(*
================================================================================
  FB_TEST_SYSTEM_VALIDATION: Test Definitivo del Sistema de Transferencia
  Versión: 1.0
  Fecha: 2026-02-21
================================================================================
  DESCRIPCIÓN:
  Test integral del core del sistema SCMTA sin dependencia de Modbus/MTZ.
  Valida la cadena completa: IO_NORMALIZE -> SCMTA -> SHED -> CMD_ARBITER -> OUTPUTS

  Simula los delays de retorno Modbus (2-4 segundos) para reproducir
  el comportamiento real de los interruptores MTZ.

  VARIABLE DE CONTROL:
  TEST_MODE:
    0 = HAPPY PATH (transferencia completa RED->GD1, retorno GD1->RED,
        failover GD1->GD2, deslastre en GD + acople, deslastre reactivo en RED)
    1 = FAULT PATH (timeout QT1, timeout QG1, timeout QT1 retorno,
        GD_ALARM arranque, GD_ALARM operación, ambos GD fallan,
        red intermitente, LOCAL bloquea)

  SIMULACIÓN MODBUS:
  Los estados de interruptores (QT1_STATE, QG1_STATE, QG2_STATE, FEEDER_STATE)
  se actualizan con un delay configurable (T_MODBUS_SIM_DELAY, default 3s)
  para simular el tiempo real que tarda Modbus RTU en reportar un cambio.

  INSTRUCCIONES:
  1. Crear instance DB "TEST_SYSTEM_DB"
  2. Setear TEST_MODE := 0 (happy) o 1 (fallas)
  3. Setear testEnable := TRUE
  4. Observar: testStep, testStatus, testResults[0..49]
  5. testReset := TRUE para reiniciar

  NOTA: Los tiempos de SCMTA se reducen para acelerar el test:
  - T_GRID_STABLE := T#5s (normalmente 120s)
  - T_GD_COOLDOWN := T#5s (normalmente 60s)
  - T_GD_READY_TIMEOUT := T#15s (normalmente 30s)
  Los tiempos de 2s (apertura/cierre interruptores) se mantienen reales.

================================================================================
*)

FUNCTION_BLOCK "FB_TEST_SYSTEM_VALIDATION"
{ S7_Optimized_Access := 'TRUE' }
VERSION : 0.1

VAR
    // ========================================================================
    // CONTROL TEST
    // ========================================================================
    testEnable : Bool := FALSE;
    testReset : Bool := FALSE;
    TEST_MODE : Int := 0;            // 0=Happy Path, 1=Fault Path
    testStep : Int := 0;
    testSubStep : Int := 0;          // Sub-paso dentro de un escenario
    testStatus : String[150] := 'Test detenido - Activar testEnable';
    testResults : Array[0..49] of Bool;  // 50 pasos de test
    testPassCount : Int := 0;        // Cantidad de tests pasados
    testFailCount : Int := 0;        // Cantidad de tests fallidos
    testTotalSteps : Int := 0;       // Total de pasos ejecutados
    testCompleted : Bool := FALSE;   // TRUE = test finalizado

    // ========================================================================
    // SIMULACIÓN MODBUS DELAY
    // ========================================================================
    T_MODBUS_SIM_DELAY : Time := T#3s; // Delay simulación respuesta Modbus

    // ========================================================================
    // SIMULACIÓN ENTRADAS FÍSICAS (para FB_IO_NORMALIZE)
    // ========================================================================
    simDI_SYS_AUTO : Bool := TRUE;
    simDI_QT1_REMOTE_SEL : Bool := TRUE;
    simDI_QT1_PB_OPEN : Bool := FALSE;
    simDI_QT1_PB_CLOSE : Bool := FALSE;
    simDI_QG1_REMOTE_SEL : Bool := TRUE;
    simDI_QG1_PB_OPEN : Bool := FALSE;
    simDI_QG1_PB_CLOSE : Bool := FALSE;
    simDI_QG2_REMOTE_SEL : Bool := TRUE;
    simDI_QG2_PB_OPEN : Bool := FALSE;
    simDI_QG2_PB_CLOSE : Bool := FALSE;
    simDI_GD_READY : Bool := FALSE;
    simDI_GD_RUNNING : Bool := FALSE;
    simDI_GD_ALARM : Bool := FALSE;
    simDI_GD2_READY : Bool := FALSE;
    simDI_GD2_RUNNING : Bool := FALSE;
    simDI_GD2_ALARM : Bool := FALSE;

    // ========================================================================
    // SIMULACIÓN ESTADOS INTERRUPTORES (respuesta Modbus simulada)
    // ========================================================================
    simQT1_STATE : Int := 1;         // 0=Abierto, 1=Cerrado, 2=Desconocido
    simQG1_STATE : Int := 0;
    simQG2_STATE : Int := 0;
    simFEEDER_STATE : Array[1..19] of Int;  // Todos inician cerrados
    simQT1_TRIPPED : Bool := FALSE;
    simQG1_TRIPPED : Bool := FALSE;
    simQG2_TRIPPED : Bool := FALSE;
    simQT1_READY : Bool := TRUE;
    simQG1_READY : Bool := TRUE;
    simQG2_READY : Bool := TRUE;
    simFEEDER_TRIPPED : Array[1..19] of Bool;
    simFEEDER_ALARM : Array[1..19] of Bool;

    // ========== Delay para simular Modbus ==========
    // Cuando CMD_ARBITER emite un CMD, el cambio de estado se aplica
    // después de T_MODBUS_SIM_DELAY (simulando la ida/vuelta Modbus)
    pendingQT1_Change : Bool := FALSE;
    pendingQT1_Target : Int := 0;
    pendingQG1_Change : Bool := FALSE;
    pendingQG1_Target : Int := 0;
    pendingQG2_Change : Bool := FALSE;
    pendingQG2_Target : Int := 0;
    pendingFeeder_Change : Array[1..19] of Bool;
    pendingFeeder_Target : Array[1..19] of Int;

    // ========================================================================
    // SIMULACIÓN MEDICIONES RED
    // ========================================================================
    simGridV_L1L2 : Real := 380.0;
    simGridV_L2L3 : Real := 380.0;
    simGridV_L3L1 : Real := 380.0;
    simGridFreq : Real := 50.0;
    simGridMeasOK : Bool := TRUE;

    // ========================================================================
    // SIMULACIÓN MEDICIONES CARGA
    // ========================================================================
    simGD_LoadPct : Real := 50.0;    // Carga GD [%]
    simTR_LoadPct : Real := 60.0;    // Carga transformador [%]

    // ========================================================================
    // SIMULACIÓN CONTROL
    // ========================================================================
    simRESET_FAULT : Bool := FALSE;

    // ========================================================================
    // VARIABLES BLOQUEO (para test de fallas)
    // ========================================================================
    blockQT1_Opening : Bool := FALSE;    // Impedir apertura QT1
    blockQG1_Closing : Bool := FALSE;    // Impedir cierre QG1
    blockQT1_Closing : Bool := FALSE;    // Impedir cierre QT1 retorno
    blockGD_Running : Bool := FALSE;     // GD1 no arranca
    blockGD_Ready : Bool := FALSE;       // GD1 no llega a READY

    // ========================================================================
    // INSTANCIAS FB (cadena completa)
    // ========================================================================
    instIO : "01_FB_IO_NORMALIZE";
    instSCMTA : "02_FB_SCMTA";
    instSHED : "03_FB_SHED";
    instARBITER : "04_FB_CMD_ARBITER";
    instOUTPUTS : "05_FB_OUTPUTS";

    // ========================================================================
    // OUTPUTS MONITOREADOS
    // ========================================================================
    // IO_NORMALIZE
    outModeAuto : Bool;
    outModeManual : Bool;
    outQT1_RemoteAllowed : Bool;
    outQG1_RemoteAllowed : Bool;
    outQG2_RemoteAllowed : Bool;
    outReqManQT1_Open : Bool;
    outReqManQT1_Close : Bool;
    outReqManQG1_Open : Bool;
    outReqManQG1_Close : Bool;
    outReqManQG2_Open : Bool;
    outReqManQG2_Close : Bool;
    outReqManFeederOpen : Array[1..19] of Bool;
    outReqManFeederClose : Array[1..19] of Bool;
    outGD_Ready : Bool;
    outGD_Running : Bool;
    outGD_Alarm : Bool;
    outGD2_Ready : Bool;
    outGD2_Running : Bool;
    outGD2_Alarm : Bool;

    // SCMTA
    outState : Int;
    outStateName : String[30];
    outReqScmtaOpenQT1 : Bool;
    outReqScmtaCloseQT1 : Bool;
    outReqScmtaOpenQG1 : Bool;
    outReqScmtaCloseQG1 : Bool;
    outReqScmtaOpenQG2 : Bool;
    outReqScmtaCloseQG2 : Bool;
    outDoGD_Start : Bool;
    outDoGD_Stop : Bool;
    outDoGD2_Start : Bool;
    outDoGD2_Stop : Bool;
    outIsOnGrid : Bool;
    outIsOnGD : Bool;
    outIsOnGD1 : Bool;
    outIsOnGD2 : Bool;
    outActiveGD : Int;
    outIsInTransfer : Bool;
    outIsFault : Bool;
    outTransferToGD : Bool;
    outGridOk : Bool;
    outGridFail : Bool;
    outFaultCode : Int;
    outElapsedTime : Time;
    outDiagLastTransferTime : Time;
    outGD1Available : Bool;
    outGD2Available : Bool;

    // SHED
    outShedReqOpen : Array[1..19] of Bool;
    outShedReqClose : Array[1..19] of Bool;
    outShedActive : Bool;
    outShedStep : Int;
    outReconnectActive : Bool;
    outReconnectStep : Int;
    outShedMode : Int;
    outFeedersShed : Int;
    outFeedersEssentialCount : Int;
    outFeedersNonEssentialCount : Int;
    outDiagLoadOverLimit : Bool;
    outDiagGdLoadOk : Bool;
    outDiagGridLoadOk : Bool;

    // CMD_ARBITER
    outCmdOpenQT1 : Bool;
    outCmdCloseQT1 : Bool;
    outCmdOpenQG1 : Bool;
    outCmdCloseQG1 : Bool;
    outCmdOpenQG2 : Bool;
    outCmdCloseQG2 : Bool;
    outCmdOpenFeeder : Array[1..19] of Bool;
    outCmdCloseFeeder : Array[1..19] of Bool;
    outBlockLocal : Bool;
    outBlockInterlock : Bool;
    outBlockConflict : Bool;
    outAlmInterlockViolation : Bool;

    // OUTPUTS
    outPilotOnGrid : Bool;
    outPilotOnGD : Bool;
    outPilotFault : Bool;
    outPilotShed : Bool;
    outAlarmBeacon : Bool;
    outHmiAlarmActive : Bool;
    outHmiAlarmText : String[100];

    // ========================================================================
    // CONFIGURACIÓN DESLASTRE (EJEMPLO: feeders 1-7 esenciales, 8-19 no-esenciales)
    // ========================================================================
    cfgFeederEssential : Array[1..19] of Bool := [TRUE, TRUE, TRUE, TRUE, TRUE, TRUE, TRUE,
                                                   FALSE, FALSE, FALSE, FALSE, FALSE, FALSE,
                                                   FALSE, FALSE, FALSE, FALSE, FALSE, FALSE];
    cfgShedEnable : Array[1..19] of Bool := [TRUE, TRUE, TRUE, TRUE, TRUE, TRUE, TRUE,
                                               TRUE, TRUE, TRUE, TRUE, TRUE, TRUE,
                                               TRUE, TRUE, TRUE, TRUE, TRUE, TRUE];
    // Orden deslastre: primero los de mayor índice (menos prioritarios)
    cfgShedOrder : Array[1..19] of Int := [19, 18, 17, 16, 15, 14, 13, 12, 11, 10, 9, 8,
                                            7, 6, 5, 4, 3, 2, 1];
    // Orden reenganche: inverso al deslastre (primero los más prioritarios)
    cfgReconnectOrder : Array[1..19] of Int := [8, 9, 10, 11, 12, 13, 14, 15, 16, 17, 18, 19,
                                                 1, 2, 3, 4, 5, 6, 7];

    // ========================================================================
    // TEMPORIZADORES TEST
    // ========================================================================
    tonStep : TON;                    // Timer general de paso
    tonModbusDelayQT1 : TON;         // Delay simulación Modbus QT1
    tonModbusDelayQG1 : TON;         // Delay simulación Modbus QG1
    tonModbusDelayQG2 : TON;         // Delay simulación Modbus QG2
    tonModbusDelayFeeder : Array[1..19] of TON; // Delay simulación feeders

    // ========================================================================
    // AUXILIARES
    // ========================================================================
    i : Int;
    initDone : Bool := FALSE;
    scenarioIndex : Int := 0;        // Escenario actual dentro del modo

END_VAR

BEGIN
    // ========================================================================
    // SECCIÓN 0: RESET
    // ========================================================================
    IF #testReset THEN
        #testStep := 0;
        #testSubStep := 0;
        #scenarioIndex := 0;
        #testStatus := 'Test reseteado';
        #testReset := FALSE;
        #testEnable := FALSE;
        #testCompleted := FALSE;
        #testPassCount := 0;
        #testFailCount := 0;
        #testTotalSteps := 0;
        #initDone := FALSE;

        // Reset condiciones
        #simQT1_STATE := 1;
        #simQG1_STATE := 0;
        #simQG2_STATE := 0;
        #simGridV_L1L2 := 380.0;
        #simGridV_L2L3 := 380.0;
        #simGridV_L3L1 := 380.0;
        #simGridFreq := 50.0;
        #simGridMeasOK := TRUE;
        #simDI_GD_READY := FALSE;
        #simDI_GD_RUNNING := FALSE;
        #simDI_GD_ALARM := FALSE;
        #simDI_GD2_READY := FALSE;
        #simDI_GD2_RUNNING := FALSE;
        #simDI_GD2_ALARM := FALSE;
        #simDI_SYS_AUTO := TRUE;
        #simDI_QT1_REMOTE_SEL := TRUE;
        #simDI_QG1_REMOTE_SEL := TRUE;
        #simDI_QG2_REMOTE_SEL := TRUE;
        #simRESET_FAULT := FALSE;
        #simGD_LoadPct := 50.0;
        #simTR_LoadPct := 60.0;
        #blockQT1_Opening := FALSE;
        #blockQG1_Closing := FALSE;
        #blockQT1_Closing := FALSE;
        #blockGD_Running := FALSE;
        #blockGD_Ready := FALSE;
        #pendingQT1_Change := FALSE;
        #pendingQG1_Change := FALSE;
        #pendingQG2_Change := FALSE;

        FOR #i := 1 TO 19 DO
            #simFEEDER_STATE[#i] := 1;  // Todos cerrados
            #simFEEDER_TRIPPED[#i] := FALSE;
            #simFEEDER_ALARM[#i] := FALSE;
            #pendingFeeder_Change[#i] := FALSE;
            #testResults[#i] := FALSE;
        END_FOR;
        FOR #i := 0 TO 49 DO
            #testResults[#i] := FALSE;
        END_FOR;

        #instSCMTA.RESET_FAULT := TRUE;
    END_IF;

    IF NOT #testEnable THEN
        RETURN;
    END_IF;


    // ========================================================================
    // SECCIÓN 1: SIMULACIÓN DELAY MODBUS (aplicar cambios pendientes)
    // Simula que el interruptor tarda T_MODBUS_SIM_DELAY en reportar
    // su nuevo estado después de recibir un comando.
    // ========================================================================

    // --- QT1 ---
    #tonModbusDelayQT1(IN := #pendingQT1_Change, PT := #T_MODBUS_SIM_DELAY);
    IF #tonModbusDelayQT1.Q AND #pendingQT1_Change THEN
        #simQT1_STATE := #pendingQT1_Target;
        #pendingQT1_Change := FALSE;
    END_IF;

    // --- QG1 ---
    #tonModbusDelayQG1(IN := #pendingQG1_Change, PT := #T_MODBUS_SIM_DELAY);
    IF #tonModbusDelayQG1.Q AND #pendingQG1_Change THEN
        #simQG1_STATE := #pendingQG1_Target;
        #pendingQG1_Change := FALSE;
    END_IF;

    // --- QG2 ---
    #tonModbusDelayQG2(IN := #pendingQG2_Change, PT := #T_MODBUS_SIM_DELAY);
    IF #tonModbusDelayQG2.Q AND #pendingQG2_Change THEN
        #simQG2_STATE := #pendingQG2_Target;
        #pendingQG2_Change := FALSE;
    END_IF;

    // --- Feeders ---
    FOR #i := 1 TO 19 DO
        #tonModbusDelayFeeder[#i](IN := #pendingFeeder_Change[#i], PT := #T_MODBUS_SIM_DELAY);
        IF #tonModbusDelayFeeder[#i].Q AND #pendingFeeder_Change[#i] THEN
            #simFEEDER_STATE[#i] := #pendingFeeder_Target[#i];
            #pendingFeeder_Change[#i] := FALSE;
        END_IF;
    END_FOR;


    // ========================================================================
    // SECCIÓN 2: CAPTURAR COMANDOS DEL ARBITER -> PROGRAMAR CAMBIO CON DELAY
    // (Solo si no hay bloqueo activo de test)
    // ========================================================================

    // QT1 Open
    IF #outCmdOpenQT1 AND NOT #blockQT1_Opening AND NOT #pendingQT1_Change THEN
        #pendingQT1_Change := TRUE;
        #pendingQT1_Target := 0;  // Abierto
    END_IF;

    // QT1 Close
    IF #outCmdCloseQT1 AND NOT #blockQT1_Closing AND NOT #pendingQT1_Change THEN
        #pendingQT1_Change := TRUE;
        #pendingQT1_Target := 1;  // Cerrado
    END_IF;

    // QG1 Open
    IF #outCmdOpenQG1 AND NOT #pendingQG1_Change THEN
        #pendingQG1_Change := TRUE;
        #pendingQG1_Target := 0;  // Abierto
    END_IF;

    // QG1 Close
    IF #outCmdCloseQG1 AND NOT #blockQG1_Closing AND NOT #pendingQG1_Change THEN
        #pendingQG1_Change := TRUE;
        #pendingQG1_Target := 1;  // Cerrado
    END_IF;

    // QG2 Open
    IF #outCmdOpenQG2 AND NOT #pendingQG2_Change THEN
        #pendingQG2_Change := TRUE;
        #pendingQG2_Target := 0;
    END_IF;

    // QG2 Close
    IF #outCmdCloseQG2 AND NOT #pendingQG2_Change THEN
        #pendingQG2_Change := TRUE;
        #pendingQG2_Target := 1;
    END_IF;

    // Feeders
    FOR #i := 1 TO 19 DO
        IF #outCmdOpenFeeder[#i] AND NOT #pendingFeeder_Change[#i] THEN
            #pendingFeeder_Change[#i] := TRUE;
            #pendingFeeder_Target[#i] := 0;  // Abierto
        END_IF;
        IF #outCmdCloseFeeder[#i] AND NOT #pendingFeeder_Change[#i] THEN
            #pendingFeeder_Change[#i] := TRUE;
            #pendingFeeder_Target[#i] := 1;  // Cerrado
        END_IF;
    END_FOR;


    // ========================================================================
    // SECCIÓN 3: EJECUTAR CADENA COMPLETA DE FBs
    // ========================================================================

    // --- FB_IO_NORMALIZE ---
    #instIO(
        DI_SYS_AUTO := #simDI_SYS_AUTO,
        DI_QT1_REMOTE_SEL := #simDI_QT1_REMOTE_SEL,
        DI_QT1_PB_OPEN := #simDI_QT1_PB_OPEN,
        DI_QT1_PB_CLOSE := #simDI_QT1_PB_CLOSE,
        DI_QG1_REMOTE_SEL := #simDI_QG1_REMOTE_SEL,
        DI_QG1_PB_OPEN := #simDI_QG1_PB_OPEN,
        DI_QG1_PB_CLOSE := #simDI_QG1_PB_CLOSE,
        DI_QG2_REMOTE_SEL := #simDI_QG2_REMOTE_SEL,
        DI_QG2_PB_OPEN := #simDI_QG2_PB_OPEN,
        DI_QG2_PB_CLOSE := #simDI_QG2_PB_CLOSE,
        DI_GD_READY := #simDI_GD_READY,
        DI_GD_RUNNING := #simDI_GD_RUNNING,
        DI_GD_ALARM := #simDI_GD_ALARM,
        DI_GD2_READY := #simDI_GD2_READY,
        DI_GD2_RUNNING := #simDI_GD2_RUNNING,
        DI_GD2_ALARM := #simDI_GD2_ALARM,

        MODE_AUTO => #outModeAuto,
        MODE_MANUAL => #outModeManual,
        QT1_REMOTE_ALLOWED => #outQT1_RemoteAllowed,
        QG1_REMOTE_ALLOWED => #outQG1_RemoteAllowed,
        QG2_REMOTE_ALLOWED => #outQG2_RemoteAllowed,
        REQ_MAN_QT1_OPEN => #outReqManQT1_Open,
        REQ_MAN_QT1_CLOSE => #outReqManQT1_Close,
        REQ_MAN_QG1_OPEN => #outReqManQG1_Open,
        REQ_MAN_QG1_CLOSE => #outReqManQG1_Close,
        REQ_MAN_QG2_OPEN => #outReqManQG2_Open,
        REQ_MAN_QG2_CLOSE => #outReqManQG2_Close,
        REQ_MAN_FEEDER_OPEN => #outReqManFeederOpen,
        REQ_MAN_FEEDER_CLOSE => #outReqManFeederClose,
        GD_READY => #outGD_Ready,
        GD_RUNNING => #outGD_Running,
        GD_ALARM => #outGD_Alarm,
        GD2_READY => #outGD2_Ready,
        GD2_RUNNING => #outGD2_Running,
        GD2_ALARM => #outGD2_Alarm
    );

    // --- FB_SCMTA ---
    #instSCMTA(
        ENABLE := TRUE,
        MODE_AUTO := #outModeAuto,
        RESET_FAULT := #simRESET_FAULT,
        QT1_STATE := #simQT1_STATE,
        QG1_STATE := #simQG1_STATE,
        QG2_STATE := #simQG2_STATE,
        GRID_V_L1L2 := #simGridV_L1L2,
        GRID_V_L2L3 := #simGridV_L2L3,
        GRID_V_L3L1 := #simGridV_L3L1,
        GRID_FREQ := #simGridFreq,
        GRID_MEASUREMENT_OK := #simGridMeasOK,
        GD_READY := #outGD_Ready,
        GD_RUNNING := #outGD_Running,
        GD_ALARM := #outGD_Alarm,
        GD2_READY := #outGD2_Ready,
        GD2_RUNNING := #outGD2_Running,
        GD2_ALARM := #outGD2_Alarm,
        // Parámetros reducidos para test
        V_NOM := 380.0,
        V_MIN_PCT := 85.0,
        V_MAX_PCT := 110.0,
        FREQ_NOM := 50.0,
        FREQ_MIN := 49.0,
        FREQ_MAX := 51.0,
        T_OPEN_QT1 := T#12s,            // Real: 2s + 3s delay Modbus + margen
        T_START_GD_DELAY := T#3s,
        T_GD_READY_TIMEOUT := T#15s,    // Reducido 30->15 para test
        T_GD_STABILIZATION := T#5s,
        T_CLOSE_QG1 := T#12s,
        T_CLOSE_QG2 := T#12s,
        T_GRID_STABLE := T#5s,          // Reducido 120->5 para test
        T_OPEN_QG1 := T#12s,
        T_OPEN_QG2 := T#12s,
        T_CLOSE_QT1 := T#12s,
        T_GD_COOLDOWN := T#5s,          // Reducido 60->5 para test
        T_GRID_FAIL_FILTER := T#2s,

        STATE => #outState,
        STATE_NAME => #outStateName,
        REQ_SCMTA_OPEN_QT1 => #outReqScmtaOpenQT1,
        REQ_SCMTA_CLOSE_QT1 => #outReqScmtaCloseQT1,
        REQ_SCMTA_OPEN_QG1 => #outReqScmtaOpenQG1,
        REQ_SCMTA_CLOSE_QG1 => #outReqScmtaCloseQG1,
        REQ_SCMTA_OPEN_QG2 => #outReqScmtaOpenQG2,
        REQ_SCMTA_CLOSE_QG2 => #outReqScmtaCloseQG2,
        DO_GD_START => #outDoGD_Start,
        DO_GD_STOP => #outDoGD_Stop,
        DO_GD2_START => #outDoGD2_Start,
        DO_GD2_STOP => #outDoGD2_Stop,
        IS_ON_GRID => #outIsOnGrid,
        IS_ON_GD => #outIsOnGD,
        IS_ON_GD1 => #outIsOnGD1,
        IS_ON_GD2 => #outIsOnGD2,
        ACTIVE_GD => #outActiveGD,
        IS_IN_TRANSFER => #outIsInTransfer,
        IS_FAULT => #outIsFault,
        TRANSFER_TO_GD => #outTransferToGD,
        GRID_OK => #outGridOk,
        GRID_FAIL => #outGridFail,
        FAULT_CODE => #outFaultCode,
        ELAPSED_TIME => #outElapsedTime,
        DIAG_LAST_TRANSFER_TIME => #outDiagLastTransferTime,
        GD1_AVAILABLE => #outGD1Available,
        GD2_AVAILABLE => #outGD2Available
    );

    // Reset pulso RESET_FAULT (1 scan)
    IF #simRESET_FAULT THEN
        #simRESET_FAULT := FALSE;
    END_IF;

    // --- FB_SHED ---
    #instSHED(
        ENABLE := TRUE,
        MODE_AUTO := #outModeAuto,
        IS_ON_GD := #outIsOnGD,
        IS_ON_GRID := #outIsOnGrid,
        IS_IN_TRANSFER := #outIsInTransfer,
        TRANSFER_TO_GD := #outTransferToGD,
        GD_LoadPct := #simGD_LoadPct,
        TR_LoadPct := #simTR_LoadPct,
        GD_SHED_ON := 90.0,
        GD_SHED_OFF := 70.0,
        GRID_SHED_ON := 85.0,
        GRID_SHED_OFF := 70.0,
        T_SHED_STEP := T#3s,           // Reducido 5->3 para test
        T_RECONNECT_STEP := T#3s,      // Reducido 5->3 para test
        T_LOAD_FILTER := T#2s,
        T_LOAD_CHECK_DELAY := T#3s,
        SHED_ORDER := #cfgShedOrder,
        RECONNECT_ORDER := #cfgReconnectOrder,
        FEEDER_ESSENTIAL := #cfgFeederEssential,
        SHED_ENABLE := #cfgShedEnable,
        FEEDER_STATE := #simFEEDER_STATE,

        REQ_SHED_OPEN => #outShedReqOpen,
        REQ_SHED_CLOSE => #outShedReqClose,
        SHED_ACTIVE => #outShedActive,
        SHED_STEP => #outShedStep,
        RECONNECT_ACTIVE => #outReconnectActive,
        RECONNECT_STEP => #outReconnectStep,
        SHED_MODE => #outShedMode,
        FEEDERS_SHED => #outFeedersShed,
        FEEDERS_ESSENTIAL_COUNT => #outFeedersEssentialCount,
        FEEDERS_NON_ESSENTIAL_COUNT => #outFeedersNonEssentialCount,
        DIAG_LOAD_OVER_LIMIT => #outDiagLoadOverLimit,
        DIAG_GD_LOAD_OK => #outDiagGdLoadOk,
        DIAG_GRID_LOAD_OK => #outDiagGridLoadOk
    );

    // --- FB_CMD_ARBITER ---
    #instARBITER(
        REQ_SCMTA_OPEN_QT1 := #outReqScmtaOpenQT1,
        REQ_SCMTA_CLOSE_QT1 := #outReqScmtaCloseQT1,
        REQ_SCMTA_OPEN_QG1 := #outReqScmtaOpenQG1,
        REQ_SCMTA_CLOSE_QG1 := #outReqScmtaCloseQG1,
        REQ_SCMTA_OPEN_QG2 := #outReqScmtaOpenQG2,
        REQ_SCMTA_CLOSE_QG2 := #outReqScmtaCloseQG2,
        REQ_SHED_OPEN := #outShedReqOpen,
        REQ_SHED_CLOSE := #outShedReqClose,
        REQ_MAN_QT1_OPEN := #outReqManQT1_Open,
        REQ_MAN_QT1_CLOSE := #outReqManQT1_Close,
        REQ_MAN_QG1_OPEN := #outReqManQG1_Open,
        REQ_MAN_QG1_CLOSE := #outReqManQG1_Close,
        REQ_MAN_QG2_OPEN := #outReqManQG2_Open,
        REQ_MAN_QG2_CLOSE := #outReqManQG2_Close,
        REQ_MAN_FEEDER_OPEN := #outReqManFeederOpen,
        REQ_MAN_FEEDER_CLOSE := #outReqManFeederClose,
        MODE_AUTO := #outModeAuto,
        MODE_MANUAL := #outModeManual,
        QT1_REMOTE_ALLOWED := #outQT1_RemoteAllowed,
        QG1_REMOTE_ALLOWED := #outQG1_RemoteAllowed,
        QG2_REMOTE_ALLOWED := #outQG2_RemoteAllowed,
        QT1_STATE := #simQT1_STATE,
        QG1_STATE := #simQG1_STATE,
        QG2_STATE := #simQG2_STATE,
        FEEDER_STATE := #simFEEDER_STATE,

        CMD_OPEN_QT1 => #outCmdOpenQT1,
        CMD_CLOSE_QT1 => #outCmdCloseQT1,
        CMD_OPEN_QG1 => #outCmdOpenQG1,
        CMD_CLOSE_QG1 => #outCmdCloseQG1,
        CMD_OPEN_QG2 => #outCmdOpenQG2,
        CMD_CLOSE_QG2 => #outCmdCloseQG2,
        CMD_OPEN_FEEDER => #outCmdOpenFeeder,
        CMD_CLOSE_FEEDER => #outCmdCloseFeeder,
        BLOCK_LOCAL => #outBlockLocal,
        BLOCK_INTERLOCK => #outBlockInterlock,
        BLOCK_CONFLICT => #outBlockConflict,
        ALM_INTERLOCK_VIOLATION => #outAlmInterlockViolation
    );

    // --- FB_OUTPUTS ---
    #instOUTPUTS(
        IS_ON_GRID := #outIsOnGrid,
        IS_ON_GD := #outIsOnGD,
        IS_IN_TRANSFER := #outIsInTransfer,
        IS_FAULT := #outIsFault,
        STATE := #outState,
        STATE_NAME := #outStateName,
        FAULT_CODE := #outFaultCode,
        QT1_STATE := #simQT1_STATE,
        QG1_STATE := #simQG1_STATE,
        QG2_STATE := #simQG2_STATE,
        QT1_TRIPPED := #simQT1_TRIPPED,
        QG1_TRIPPED := #simQG1_TRIPPED,
        QG2_TRIPPED := #simQG2_TRIPPED,
        QT1_READY := #simQT1_READY,
        QG1_READY := #simQG1_READY,
        QG2_READY := #simQG2_READY,
        FEEDER_STATE := #simFEEDER_STATE,
        FEEDER_TRIPPED := #simFEEDER_TRIPPED,
        FEEDER_ALARM := #simFEEDER_ALARM,
        ALM_INTERLOCK_VIOLATION := #outAlmInterlockViolation,
        BLOCK_INTERLOCK := #outBlockInterlock,
        GRID_FAIL := #outGridFail,
        GD_ALARM := #outGD_Alarm,
        GD2_ALARM := #outGD2_Alarm,
        SHED_ACTIVE := #outShedActive,
        FEEDERS_SHED := #outFeedersShed,
        ACK_ALARM := FALSE,

        DO_PILOT_ON_GRID => #outPilotOnGrid,
        DO_PILOT_ON_GD => #outPilotOnGD,
        DO_PILOT_FAULT => #outPilotFault,
        DO_PILOT_SHED => #outPilotShed,
        DO_ALARM_BEACON => #outAlarmBeacon,
        HMI_ALARM_ACTIVE => #outHmiAlarmActive,
        HMI_ALARM_TEXT => #outHmiAlarmText
    );


    // ========================================================================
    // SECCIÓN 4: SECUENCIA DE TEST SEGÚN TEST_MODE
    // ========================================================================

    IF #TEST_MODE = 0 THEN
        // ====================================================================
        // =================== HAPPY PATH (TEST_MODE = 0) =====================
        // ====================================================================

        CASE #testStep OF

            // ================================================================
            // ESCENARIO A: TRANSFERENCIA RED -> GD1 COMPLETA
            // ================================================================

            // PASO 0: Verificar estado inicial NORMAL_ON_GRID
            0:
                #testStatus := 'HP-00: Init - Verificar NORMAL_ON_GRID';
                #tonStep(IN := TRUE, PT := T#5s);
                IF #tonStep.Q THEN
                    #testResults[0] := (#outState = 1) AND #outIsOnGrid AND NOT #outIsOnGD
                                       AND #outPilotOnGrid AND NOT #outPilotOnGD
                                       AND NOT #outPilotFault;
                    IF #testResults[0] THEN #testPassCount := #testPassCount + 1;
                    ELSE #testFailCount := #testFailCount + 1; END_IF;
                    #testTotalSteps := #testTotalSteps + 1;
                    #tonStep(IN := FALSE, PT := T#1s);
                    #testStep := 1;
                END_IF;

            // PASO 1: Simular falla de RED -> detectar GRID_FAIL
            1:
                #testStatus := 'HP-01: Falla RED - Esperar GRID_FAIL_DETECTED';
                #simGridV_L1L2 := 200.0;
                #simGridV_L2L3 := 200.0;
                #simGridV_L3L1 := 200.0;
                #simGridFreq := 48.0;

                #tonStep(IN := TRUE, PT := T#5s);
                IF #tonStep.Q THEN
                    #testResults[1] := (#outState >= 2) AND #outGridFail
                                       AND #outIsInTransfer;
                    IF #testResults[1] THEN #testPassCount := #testPassCount + 1;
                    ELSE #testFailCount := #testFailCount + 1; END_IF;
                    #testTotalSteps := #testTotalSteps + 1;
                    #tonStep(IN := FALSE, PT := T#1s);
                    #testStep := 2;
                END_IF;

            // PASO 2: Verificar OPEN_QT1 + TRANSFER_TO_GD + señal SHED desacople
            2:
                #testStatus := 'HP-02: OPEN_QT1 - QT1 abre con delay Modbus';
                #tonStep(IN := TRUE, PT := T#8s);  // 3s SCMTA + 3s delay Modbus + margen
                IF #simQT1_STATE = 0 THEN
                    // QT1 se abrió (después del delay Modbus)
                    #testResults[2] := (#outState >= 3) AND #outTransferToGD;
                    IF #testResults[2] THEN #testPassCount := #testPassCount + 1;
                    ELSE #testFailCount := #testFailCount + 1; END_IF;
                    #testTotalSteps := #testTotalSteps + 1;
                    #tonStep(IN := FALSE, PT := T#1s);
                    #testStep := 3;
                ELSIF #tonStep.Q THEN
                    // Timeout: QT1 no abrió
                    #testResults[2] := FALSE;
                    #testFailCount := #testFailCount + 1;
                    #testTotalSteps := #testTotalSteps + 1;
                    #tonStep(IN := FALSE, PT := T#1s);
                    #testStep := 3;
                END_IF;

            // PASO 3: GD1 arranca -> simular GD_RUNNING
            3:
                #testStatus := 'HP-03: START_GD1 - Simular arranque GD1';
                // Esperar que SCMTA pida arranque
                IF #outDoGD_Start THEN
                    #simDI_GD_RUNNING := TRUE;
                END_IF;

                #tonStep(IN := TRUE, PT := T#8s);
                IF #tonStep.Q THEN
                    #testResults[3] := #outDoGD_Start OR #simDI_GD_RUNNING;
                    IF #testResults[3] THEN #testPassCount := #testPassCount + 1;
                    ELSE #testFailCount := #testFailCount + 1; END_IF;
                    #testTotalSteps := #testTotalSteps + 1;
                    #tonStep(IN := FALSE, PT := T#1s);
                    #testStep := 4;
                END_IF;

            // PASO 4: GD1 listo -> simular GD_READY + estabilización -> CLOSE_QG1
            4:
                #testStatus := 'HP-04: WAIT_GD1_READY - Simular GD1 listo';
                #simDI_GD_Ready := TRUE;

                #tonStep(IN := TRUE, PT := T#10s);  // 5s estab + margen
                IF #outState = 7 OR #simQG1_STATE = 1 THEN
                    // Llegó a CLOSE_QG1 o QG1 ya cerró con delay
                    #testResults[4] := TRUE;
                    IF #testResults[4] THEN #testPassCount := #testPassCount + 1;
                    ELSE #testFailCount := #testFailCount + 1; END_IF;
                    #testTotalSteps := #testTotalSteps + 1;
                    #tonStep(IN := FALSE, PT := T#1s);
                    #testStep := 5;
                ELSIF #tonStep.Q THEN
                    #testResults[4] := FALSE;
                    #testFailCount := #testFailCount + 1;
                    #testTotalSteps := #testTotalSteps + 1;
                    #tonStep(IN := FALSE, PT := T#1s);
                    #testStep := 5;
                END_IF;

            // PASO 5: Verificar ON_GD1 + pilotos
            5:
                #testStatus := 'HP-05: ON_GD1 - Verificar operación con GD1';
                #tonStep(IN := TRUE, PT := T#8s);
                IF #outState = 8 THEN
                    #testResults[5] := #outIsOnGD AND #outIsOnGD1 AND NOT #outIsOnGrid
                                       AND (#outActiveGD = 1) AND NOT #outIsInTransfer
                                       AND #outPilotOnGD AND NOT #outPilotOnGrid;
                    IF #testResults[5] THEN #testPassCount := #testPassCount + 1;
                    ELSE #testFailCount := #testFailCount + 1; END_IF;
                    #testTotalSteps := #testTotalSteps + 1;
                    #tonStep(IN := FALSE, PT := T#1s);
                    #testStep := 6;
                ELSIF #tonStep.Q THEN
                    #testResults[5] := FALSE;
                    #testFailCount := #testFailCount + 1;
                    #testTotalSteps := #testTotalSteps + 1;
                    #tonStep(IN := FALSE, PT := T#1s);
                    #testStep := 6;
                END_IF;

            // ================================================================
            // ESCENARIO B: DESLASTRE EN GD + ACOPLE ESCALONADO
            // ================================================================

            // PASO 6: Verificar que SHED desacopló no-esenciales
            6:
                #testStatus := 'HP-06: SHED - Verificar no-esenciales desacoplados';
                #tonStep(IN := TRUE, PT := T#5s);
                IF #tonStep.Q THEN
                    // Feeders 8-19 (no-esenciales) deben estar abiertos
                    // Feeders 1-7 (esenciales) deben seguir cerrados
                    #testResults[6] := (#simFEEDER_STATE[1] = 1) AND
                                       (#simFEEDER_STATE[7] = 1);
                    // Al menos algunos no-esenciales abiertos
                    IF #outFeedersShed > 0 THEN
                        #testResults[6] := #testResults[6] AND TRUE;
                    END_IF;
                    IF #testResults[6] THEN #testPassCount := #testPassCount + 1;
                    ELSE #testFailCount := #testFailCount + 1; END_IF;
                    #testTotalSteps := #testTotalSteps + 1;
                    #tonStep(IN := FALSE, PT := T#1s);
                    #testStep := 7;
                END_IF;

            // PASO 7: Verificar acoplamiento escalonado comienza (carga OK)
            7:
                #testStatus := 'HP-07: SHED - Acoplamiento escalonado en GD';
                #simGD_LoadPct := 50.0;  // Carga baja, permite acoplar

                #tonStep(IN := TRUE, PT := T#15s);  // Tiempo para varios pasos
                IF #tonStep.Q THEN
                    // Verificar que al menos un feeder no-esencial se reacopló
                    #testResults[7] := (#outShedMode = 3) OR   // GD_RECONNECT
                                       (#outReconnectStep > 0) OR
                                       (#outFeedersShed < 12);  // Menos de 12 abiertos
                    IF #testResults[7] THEN #testPassCount := #testPassCount + 1;
                    ELSE #testFailCount := #testFailCount + 1; END_IF;
                    #testTotalSteps := #testTotalSteps + 1;
                    #tonStep(IN := FALSE, PT := T#1s);
                    #testStep := 8;
                END_IF;

            // PASO 8: Subir carga GD -> verificar que SHED reactivo frena acople
            8:
                #testStatus := 'HP-08: SHED - Carga GD sube, freno acoplamiento';
                #simGD_LoadPct := 92.0;  // Sobre umbral GD_SHED_ON (90%)

                #tonStep(IN := TRUE, PT := T#8s);
                IF #tonStep.Q THEN
                    #testResults[8] := #outDiagLoadOverLimit OR #outShedActive OR
                                       NOT #outReconnectActive;
                    IF #testResults[8] THEN #testPassCount := #testPassCount + 1;
                    ELSE #testFailCount := #testFailCount + 1; END_IF;
                    #testTotalSteps := #testTotalSteps + 1;
                    #simGD_LoadPct := 50.0;  // Restaurar carga normal
                    #tonStep(IN := FALSE, PT := T#1s);
                    #testStep := 9;
                END_IF;

            // ================================================================
            // ESCENARIO C: RETORNO GD1 -> RED
            // ================================================================

            // PASO 9: Restaurar RED -> detectar GRID_RETURN
            9:
                #testStatus := 'HP-09: Restaurar RED - Esperar GRID_RETURN';
                #simGridV_L1L2 := 380.0;
                #simGridV_L2L3 := 380.0;
                #simGridV_L3L1 := 380.0;
                #simGridFreq := 50.0;

                #tonStep(IN := TRUE, PT := T#8s);
                IF #outState = 9 OR #outState = 10 THEN
                    #testResults[9] := TRUE;
                    #testPassCount := #testPassCount + 1;
                    #testTotalSteps := #testTotalSteps + 1;
                    #tonStep(IN := FALSE, PT := T#1s);
                    #testStep := 10;
                ELSIF #tonStep.Q THEN
                    #testResults[9] := FALSE;
                    #testFailCount := #testFailCount + 1;
                    #testTotalSteps := #testTotalSteps + 1;
                    #tonStep(IN := FALSE, PT := T#1s);
                    #testStep := 10;
                END_IF;

            // PASO 10: Esperar red estable 5s -> OPEN_QG1 -> CLOSE_QT1
            10:
                #testStatus := 'HP-10: WAIT_GRID_STABLE + retorno a RED';
                #tonStep(IN := TRUE, PT := T#20s);  // 5s estable + delay open/close + margen

                IF #outState = 1 THEN
                    // Volvió a NORMAL_ON_GRID
                    #testResults[10] := #outIsOnGrid AND NOT #outIsOnGD
                                        AND #outPilotOnGrid AND NOT #outPilotOnGD;
                    IF #testResults[10] THEN #testPassCount := #testPassCount + 1;
                    ELSE #testFailCount := #testFailCount + 1; END_IF;
                    #testTotalSteps := #testTotalSteps + 1;
                    #tonStep(IN := FALSE, PT := T#1s);
                    #testStep := 11;
                ELSIF #tonStep.Q THEN
                    #testResults[10] := FALSE;
                    #testFailCount := #testFailCount + 1;
                    #testTotalSteps := #testTotalSteps + 1;
                    #tonStep(IN := FALSE, PT := T#1s);
                    #testStep := 11;
                END_IF;

            // PASO 11: Verificar GD_STOP después del cooldown
            11:
                #testStatus := 'HP-11: GD_COOLDOWN - Verificar parada GD1';
                #tonStep(IN := TRUE, PT := T#3s);
                IF #tonStep.Q THEN
                    // El GD debería haber recibido orden de parada
                    #testResults[11] := (#outState = 1);
                    IF #testResults[11] THEN #testPassCount := #testPassCount + 1;
                    ELSE #testFailCount := #testFailCount + 1; END_IF;
                    #testTotalSteps := #testTotalSteps + 1;
                    #tonStep(IN := FALSE, PT := T#1s);
                    // Reiniciar GD a idle
                    #simDI_GD_RUNNING := FALSE;
                    #simDI_GD_Ready := FALSE;
                    #testStep := 12;
                END_IF;

            // ================================================================
            // ESCENARIO D: FAILOVER GD1 -> GD2
            // ================================================================

            // PASO 12: Nueva falla RED
            12:
                #testStatus := 'HP-12: FAILOVER - Nueva falla RED';
                #simGridV_L1L2 := 200.0;
                #simGridV_L2L3 := 200.0;
                #simGridV_L3L1 := 200.0;

                #tonStep(IN := TRUE, PT := T#5s);
                IF #outState >= 2 THEN
                    #testResults[12] := TRUE;
                    #testPassCount := #testPassCount + 1;
                    #testTotalSteps := #testTotalSteps + 1;
                    #tonStep(IN := FALSE, PT := T#1s);
                    #testStep := 13;
                ELSIF #tonStep.Q THEN
                    #testResults[12] := FALSE;
                    #testFailCount := #testFailCount + 1;
                    #testTotalSteps := #testTotalSteps + 1;
                    #tonStep(IN := FALSE, PT := T#1s);
                    #testStep := 13;
                END_IF;

            // PASO 13: GD1 falla durante arranque -> failover a GD2
            13:
                #testStatus := 'HP-13: FAILOVER - GD1 ALARM durante arranque';
                // Esperar que SCMTA intente arrancar GD1
                IF #outState = 5 OR #outDoGD_Start THEN
                    #simDI_GD_ALARM := TRUE;  // GD1 falla
                END_IF;

                #tonStep(IN := TRUE, PT := T#10s);
                IF #outState = 15 OR #outState = 16 OR #outState = 17 THEN
                    // Pasó a camino GD2 (START_GD2_DELAY, START_GD2, o WAIT_GD2_READY)
                    #testResults[13] := TRUE;
                    #testPassCount := #testPassCount + 1;
                    #testTotalSteps := #testTotalSteps + 1;
                    #tonStep(IN := FALSE, PT := T#1s);
                    #testStep := 14;
                ELSIF #tonStep.Q THEN
                    #testResults[13] := FALSE;
                    #testFailCount := #testFailCount + 1;
                    #testTotalSteps := #testTotalSteps + 1;
                    #tonStep(IN := FALSE, PT := T#1s);
                    #testStep := 14;
                END_IF;

            // PASO 14: GD2 arranca y llega a ON_GD2
            14:
                #testStatus := 'HP-14: FAILOVER - GD2 arranca -> ON_GD2';
                IF #outDoGD2_Start THEN
                    #simDI_GD2_RUNNING := TRUE;
                END_IF;
                #simDI_GD2_Ready := TRUE;

                #tonStep(IN := TRUE, PT := T#15s);
                IF #outState = 19 THEN
                    // ON_GD2
                    #testResults[14] := #outIsOnGD2 AND (#outActiveGD = 2)
                                        AND NOT #outIsFault;
                    IF #testResults[14] THEN #testPassCount := #testPassCount + 1;
                    ELSE #testFailCount := #testFailCount + 1; END_IF;
                    #testTotalSteps := #testTotalSteps + 1;
                    #tonStep(IN := FALSE, PT := T#1s);
                    #testStep := 15;
                ELSIF #tonStep.Q THEN
                    #testResults[14] := FALSE;
                    #testFailCount := #testFailCount + 1;
                    #testTotalSteps := #testTotalSteps + 1;
                    #tonStep(IN := FALSE, PT := T#1s);
                    #testStep := 15;
                END_IF;

            // ================================================================
            // ESCENARIO E: DESLASTRE REACTIVO EN RED
            // ================================================================

            // PASO 15: Retorno a RED desde GD2 para probar deslastre RED
            15:
                #testStatus := 'HP-15: Restaurar RED desde GD2';
                #simGridV_L1L2 := 380.0;
                #simGridV_L2L3 := 380.0;
                #simGridV_L3L1 := 380.0;
                #simGridFreq := 50.0;

                #tonStep(IN := TRUE, PT := T#25s);  // Esperar retorno completo
                IF #outState = 1 THEN
                    #testResults[15] := #outIsOnGrid;
                    IF #testResults[15] THEN #testPassCount := #testPassCount + 1;
                    ELSE #testFailCount := #testFailCount + 1; END_IF;
                    #testTotalSteps := #testTotalSteps + 1;
                    #tonStep(IN := FALSE, PT := T#1s);
                    #simDI_GD_ALARM := FALSE;
                    #simDI_GD2_RUNNING := FALSE;
                    #simDI_GD2_Ready := FALSE;
                    // Asegurar feeders cerrados para test
                    FOR #i := 1 TO 19 DO
                        #simFEEDER_STATE[#i] := 1;
                    END_FOR;
                    #testStep := 16;
                ELSIF #tonStep.Q THEN
                    #testResults[15] := FALSE;
                    #testFailCount := #testFailCount + 1;
                    #testTotalSteps := #testTotalSteps + 1;
                    #tonStep(IN := FALSE, PT := T#1s);
                    #testStep := 16;
                END_IF;

            // PASO 16: Sobrecarga transformador -> deslastre reactivo en RED
            16:
                #testStatus := 'HP-16: Sobrecarga trafo -> deslastre reactivo RED';
                #simTR_LoadPct := 88.0;  // Sobre GRID_SHED_ON (85%)

                #tonStep(IN := TRUE, PT := T#15s);
                IF #tonStep.Q THEN
                    #testResults[16] := (#outShedMode = 1) OR #outShedActive OR
                                        (#outFeedersShed > 0);
                    IF #testResults[16] THEN #testPassCount := #testPassCount + 1;
                    ELSE #testFailCount := #testFailCount + 1; END_IF;
                    #testTotalSteps := #testTotalSteps + 1;
                    #tonStep(IN := FALSE, PT := T#1s);
                    #testStep := 17;
                END_IF;

            // PASO 17: Bajar carga -> histéresis -> reenganche en RED
            17:
                #testStatus := 'HP-17: Carga baja -> reenganche en RED (histeresis)';
                #simTR_LoadPct := 65.0;  // Bajo GRID_SHED_OFF (70%)

                #tonStep(IN := TRUE, PT := T#15s);
                IF #tonStep.Q THEN
                    #testResults[17] := (#outShedMode = 5) OR    // GRID_RECONNECT
                                        #outReconnectActive OR
                                        NOT #outShedActive;
                    IF #testResults[17] THEN #testPassCount := #testPassCount + 1;
                    ELSE #testFailCount := #testFailCount + 1; END_IF;
                    #testTotalSteps := #testTotalSteps + 1;
                    #tonStep(IN := FALSE, PT := T#1s);
                    #simTR_LoadPct := 60.0;
                    #testStep := 18;
                END_IF;

            // PASO 18: HAPPY PATH COMPLETADO
            18:
                #testStatus := 'HP COMPLETADO - Pass:' ;
                #testCompleted := TRUE;
                // Test terminado

        END_CASE;  // Fin HAPPY PATH


    ELSIF #TEST_MODE = 1 THEN
        // ====================================================================
        // =================== FAULT PATH (TEST_MODE = 1) =====================
        // ====================================================================

        CASE #testStep OF

            // ================================================================
            // ESCENARIO F: TIMEOUT QT1 NO ABRE
            // ================================================================

            // PASO 0: Init estado NORMAL_ON_GRID
            0:
                #testStatus := 'FP-00: Init NORMAL_ON_GRID para test fallas';
                #simQT1_STATE := 1;
                #simQG1_STATE := 0;
                #simQG2_STATE := 0;
                #simGridV_L1L2 := 380.0;
                #simGridV_L2L3 := 380.0;
                #simGridV_L3L1 := 380.0;
                #simGridFreq := 50.0;
                #blockQT1_Opening := FALSE;
                #blockQG1_Closing := FALSE;
                #blockQT1_Closing := FALSE;

                #tonStep(IN := TRUE, PT := T#5s);
                IF #tonStep.Q THEN
                    #testResults[0] := (#outState = 1);
                    IF #testResults[0] THEN #testPassCount := #testPassCount + 1;
                    ELSE #testFailCount := #testFailCount + 1; END_IF;
                    #testTotalSteps := #testTotalSteps + 1;
                    #tonStep(IN := FALSE, PT := T#1s);
                    #testStep := 1;
                END_IF;

            // PASO 1: Falla RED + BLOQUEAR apertura QT1 -> timeout
            1:
                #testStatus := 'FP-01: Falla RED - QT1 BLOQUEADO (no abre)';
                #simGridV_L1L2 := 200.0;
                #simGridV_L2L3 := 200.0;
                #simGridV_L3L1 := 200.0;
                #blockQT1_Opening := TRUE;
                #simQT1_STATE := 1;  // Forzar cerrado (bloqueo actúa en SECCIÓN 2)
                // Cancelar pending
                #pendingQT1_Change := FALSE;

                #tonStep(IN := TRUE, PT := T#18s);  // T_OPEN_QT1=12s + margen
                IF #outState = 14 THEN
                    // FAULT_LOCKOUT
                    #testResults[1] := #outIsFault AND (#outFaultCode = 101);
                    IF #testResults[1] THEN #testPassCount := #testPassCount + 1;
                    ELSE #testFailCount := #testFailCount + 1; END_IF;
                    #testTotalSteps := #testTotalSteps + 1;
                    #tonStep(IN := FALSE, PT := T#1s);
                    #testStep := 2;
                ELSIF #tonStep.Q THEN
                    #testResults[1] := FALSE;
                    #testFailCount := #testFailCount + 1;
                    #testTotalSteps := #testTotalSteps + 1;
                    #tonStep(IN := FALSE, PT := T#1s);
                    #testStep := 2;
                END_IF;

            // PASO 2: Verificar pilotos FAULT + reset
            2:
                #testStatus := 'FP-02: Verificar FAULT_LOCKOUT + reset';
                #testResults[2] := #outPilotFault AND #outIsFault;
                IF #testResults[2] THEN #testPassCount := #testPassCount + 1;
                ELSE #testFailCount := #testFailCount + 1; END_IF;
                #testTotalSteps := #testTotalSteps + 1;

                // Reset fault
                #blockQT1_Opening := FALSE;
                #simGridV_L1L2 := 380.0;
                #simGridV_L2L3 := 380.0;
                #simGridV_L3L1 := 380.0;
                #simGridFreq := 50.0;
                #simQT1_STATE := 1;
                #simRESET_FAULT := TRUE;
                #testStep := 3;

            // PASO 3: Esperar recuperación post-reset
            3:
                #testStatus := 'FP-03: Esperar recuperacion post-reset';
                #tonStep(IN := TRUE, PT := T#5s);
                IF #tonStep.Q THEN
                    #testResults[3] := (#outState = 1) AND NOT #outIsFault;
                    IF #testResults[3] THEN #testPassCount := #testPassCount + 1;
                    ELSE #testFailCount := #testFailCount + 1; END_IF;
                    #testTotalSteps := #testTotalSteps + 1;
                    #tonStep(IN := FALSE, PT := T#1s);
                    #testStep := 4;
                END_IF;

            // ================================================================
            // ESCENARIO G: TIMEOUT QG1 NO CIERRA
            // ================================================================

            // PASO 4: Falla RED + QT1 abre OK + GD1 arranca + QG1 BLOQUEADO
            4:
                #testStatus := 'FP-04: Falla RED - QG1 BLOQUEADO (no cierra)';
                #simGridV_L1L2 := 200.0;
                #simGridV_L2L3 := 200.0;
                #simGridV_L3L1 := 200.0;
                #blockQG1_Closing := TRUE;

                // Simular GD1 arranque normal
                IF #outDoGD_Start THEN
                    #simDI_GD_RUNNING := TRUE;
                END_IF;
                IF #outState >= 6 THEN
                    #simDI_GD_Ready := TRUE;
                END_IF;

                // Cancelar cierre QG1 pendiente
                IF #pendingQG1_Change AND #pendingQG1_Target = 1 THEN
                    #pendingQG1_Change := FALSE;
                END_IF;

                #tonStep(IN := TRUE, PT := T#30s);  // GD_READY_TIMEOUT + margen
                IF #outState = 14 THEN
                    #testResults[4] := #outIsFault AND (#outFaultCode = 103);
                    IF #testResults[4] THEN #testPassCount := #testPassCount + 1;
                    ELSE #testFailCount := #testFailCount + 1; END_IF;
                    #testTotalSteps := #testTotalSteps + 1;
                    #tonStep(IN := FALSE, PT := T#1s);
                    #testStep := 5;
                ELSIF #tonStep.Q THEN
                    #testResults[4] := FALSE;
                    #testFailCount := #testFailCount + 1;
                    #testTotalSteps := #testTotalSteps + 1;
                    #tonStep(IN := FALSE, PT := T#1s);
                    #testStep := 5;
                END_IF;

            // PASO 5: Reset y recuperar
            5:
                #testStatus := 'FP-05: Reset post QG1 timeout';
                #blockQG1_Closing := FALSE;
                #simGridV_L1L2 := 380.0;
                #simGridV_L2L3 := 380.0;
                #simGridV_L3L1 := 380.0;
                #simQT1_STATE := 1;
                #simQG1_STATE := 0;
                #simDI_GD_RUNNING := FALSE;
                #simDI_GD_Ready := FALSE;
                #simRESET_FAULT := TRUE;

                #tonStep(IN := TRUE, PT := T#5s);
                IF #tonStep.Q THEN
                    #testResults[5] := NOT #outIsFault;
                    IF #testResults[5] THEN #testPassCount := #testPassCount + 1;
                    ELSE #testFailCount := #testFailCount + 1; END_IF;
                    #testTotalSteps := #testTotalSteps + 1;
                    #tonStep(IN := FALSE, PT := T#1s);
                    #testStep := 6;
                END_IF;

            // ================================================================
            // ESCENARIO H: GD_ALARM DURANTE ARRANQUE -> FAILOVER GD2
            // ================================================================

            // PASO 6: Falla RED + GD1 ALARM durante START
            6:
                #testStatus := 'FP-06: GD1 ALARM arranque -> failover GD2';
                #simGridV_L1L2 := 200.0;
                #simGridV_L2L3 := 200.0;
                #simGridV_L3L1 := 200.0;

                IF #outState = 5 OR #outDoGD_Start THEN
                    #simDI_GD_ALARM := TRUE;
                END_IF;

                #tonStep(IN := TRUE, PT := T#15s);
                IF #outState >= 15 AND #outState <= 18 THEN
                    #testResults[6] := TRUE;  // Pasó a camino GD2
                    #testPassCount := #testPassCount + 1;
                    #testTotalSteps := #testTotalSteps + 1;
                    #tonStep(IN := FALSE, PT := T#1s);
                    #testStep := 7;
                ELSIF #tonStep.Q THEN
                    #testResults[6] := FALSE;
                    #testFailCount := #testFailCount + 1;
                    #testTotalSteps := #testTotalSteps + 1;
                    #tonStep(IN := FALSE, PT := T#1s);
                    #testStep := 7;
                END_IF;

            // ================================================================
            // ESCENARIO I: AMBOS GD FALLAN -> FAULT_LOCKOUT (209)
            // ================================================================

            // PASO 7: GD2 también alarma -> ambos fallan
            7:
                #testStatus := 'FP-07: GD2 ALARM -> AMBOS GD FALLAN -> LOCKOUT';
                #simDI_GD2_ALARM := TRUE;  // GD2 también falla

                #tonStep(IN := TRUE, PT := T#15s);
                IF #outState = 14 THEN
                    #testResults[7] := #outIsFault AND (#outFaultCode = 209);
                    IF #testResults[7] THEN #testPassCount := #testPassCount + 1;
                    ELSE #testFailCount := #testFailCount + 1; END_IF;
                    #testTotalSteps := #testTotalSteps + 1;
                    #tonStep(IN := FALSE, PT := T#1s);
                    #testStep := 8;
                ELSIF #tonStep.Q THEN
                    #testResults[7] := FALSE;
                    #testFailCount := #testFailCount + 1;
                    #testTotalSteps := #testTotalSteps + 1;
                    #tonStep(IN := FALSE, PT := T#1s);
                    #testStep := 8;
                END_IF;

            // PASO 8: Reset + recuperar
            8:
                #testStatus := 'FP-08: Reset post ambos GD';
                #simDI_GD_ALARM := FALSE;
                #simDI_GD2_ALARM := FALSE;
                #simGridV_L1L2 := 380.0;
                #simGridV_L2L3 := 380.0;
                #simGridV_L3L1 := 380.0;
                #simQT1_STATE := 1;
                #simQG1_STATE := 0;
                #simQG2_STATE := 0;
                #simRESET_FAULT := TRUE;

                #tonStep(IN := TRUE, PT := T#5s);
                IF #tonStep.Q THEN
                    #testResults[8] := NOT #outIsFault;
                    IF #testResults[8] THEN #testPassCount := #testPassCount + 1;
                    ELSE #testFailCount := #testFailCount + 1; END_IF;
                    #testTotalSteps := #testTotalSteps + 1;
                    #tonStep(IN := FALSE, PT := T#1s);
                    #testStep := 9;
                END_IF;

            // ================================================================
            // ESCENARIO J: GD_ALARM DURANTE OPERACIÓN (ON_GD1) -> FAILOVER
            // ================================================================

            // PASO 9: Falla RED + transferir a GD1 normalmente
            9:
                #testStatus := 'FP-09: Transferir a GD1 para test alarm en operacion';
                #simGridV_L1L2 := 200.0;
                #simGridV_L2L3 := 200.0;
                #simGridV_L3L1 := 200.0;

                IF #outDoGD_Start THEN
                    #simDI_GD_RUNNING := TRUE;
                END_IF;
                IF #outState >= 6 THEN
                    #simDI_GD_Ready := TRUE;
                END_IF;

                #tonStep(IN := TRUE, PT := T#20s);
                IF #outState = 8 THEN
                    #testResults[9] := #outIsOnGD1;
                    IF #testResults[9] THEN #testPassCount := #testPassCount + 1;
                    ELSE #testFailCount := #testFailCount + 1; END_IF;
                    #testTotalSteps := #testTotalSteps + 1;
                    #tonStep(IN := FALSE, PT := T#1s);
                    #testStep := 10;
                ELSIF #tonStep.Q THEN
                    #testResults[9] := FALSE;
                    #testFailCount := #testFailCount + 1;
                    #testTotalSteps := #testTotalSteps + 1;
                    #tonStep(IN := FALSE, PT := T#1s);
                    #testStep := 10;
                END_IF;

            // PASO 10: GD1 ALARM en operación -> failover a GD2
            10:
                #testStatus := 'FP-10: GD1 ALARM en ON_GD1 -> OPEN_GD_FOR_SWITCH';
                #simDI_GD_ALARM := TRUE;

                #tonStep(IN := TRUE, PT := T#10s);
                IF #outState = 20 OR (#outState >= 15 AND #outState <= 18) THEN
                    #testResults[10] := TRUE;
                    #testPassCount := #testPassCount + 1;
                    #testTotalSteps := #testTotalSteps + 1;
                    #tonStep(IN := FALSE, PT := T#1s);
                    #testStep := 11;
                ELSIF #tonStep.Q THEN
                    #testResults[10] := FALSE;
                    #testFailCount := #testFailCount + 1;
                    #testTotalSteps := #testTotalSteps + 1;
                    #tonStep(IN := FALSE, PT := T#1s);
                    #testStep := 11;
                END_IF;

            // PASO 11: GD2 arranca -> ON_GD2
            11:
                #testStatus := 'FP-11: GD2 asume carga -> ON_GD2';
                IF #outDoGD2_Start THEN
                    #simDI_GD2_RUNNING := TRUE;
                END_IF;
                #simDI_GD2_Ready := TRUE;

                #tonStep(IN := TRUE, PT := T#15s);
                IF #outState = 19 THEN
                    #testResults[11] := #outIsOnGD2;
                    IF #testResults[11] THEN #testPassCount := #testPassCount + 1;
                    ELSE #testFailCount := #testFailCount + 1; END_IF;
                    #testTotalSteps := #testTotalSteps + 1;
                    #tonStep(IN := FALSE, PT := T#1s);
                    #testStep := 12;
                ELSIF #tonStep.Q THEN
                    #testResults[11] := FALSE;
                    #testFailCount := #testFailCount + 1;
                    #testTotalSteps := #testTotalSteps + 1;
                    #tonStep(IN := FALSE, PT := T#1s);
                    #testStep := 12;
                END_IF;

            // ================================================================
            // ESCENARIO K: RED INTERMITENTE DURANTE WAIT_GRID_STABLE
            // ================================================================

            // PASO 12: Restaurar RED -> detectar retorno -> luego falla de nuevo
            12:
                #testStatus := 'FP-12: RED intermitente durante WAIT_GRID_STABLE';
                #simGridV_L1L2 := 380.0;
                #simGridV_L2L3 := 380.0;
                #simGridV_L3L1 := 380.0;

                #tonStep(IN := TRUE, PT := T#5s);
                IF #outState = 10 THEN
                    // Está esperando red estable -> forzar falla de nuevo
                    #simGridV_L1L2 := 200.0;
                    #simGridV_L2L3 := 200.0;
                    #simGridV_L3L1 := 200.0;
                END_IF;

                IF #tonStep.Q THEN
                    // Debería haber vuelto a ON_GD2 (no completó estabilidad)
                    #testResults[12] := (#outState = 19) OR (#outState = 8);
                    IF #testResults[12] THEN #testPassCount := #testPassCount + 1;
                    ELSE #testFailCount := #testFailCount + 1; END_IF;
                    #testTotalSteps := #testTotalSteps + 1;
                    #tonStep(IN := FALSE, PT := T#1s);
                    #testStep := 13;
                END_IF;

            // ================================================================
            // ESCENARIO L: SELECTOR LOCAL BLOQUEA COMANDOS
            // ================================================================

            // PASO 13: Reset y preparar test LOCAL
            13:
                #testStatus := 'FP-13: Preparar test LOCAL/REMOTO';
                #simGridV_L1L2 := 380.0;
                #simGridV_L2L3 := 380.0;
                #simGridV_L3L1 := 380.0;
                #simDI_GD_ALARM := FALSE;
                #simDI_GD2_ALARM := FALSE;
                #simDI_GD_RUNNING := FALSE;
                #simDI_GD2_RUNNING := FALSE;
                #simDI_GD_Ready := FALSE;
                #simDI_GD2_Ready := FALSE;
                #simQT1_STATE := 1;
                #simQG1_STATE := 0;
                #simQG2_STATE := 0;
                #simRESET_FAULT := TRUE;

                #tonStep(IN := TRUE, PT := T#5s);
                IF #tonStep.Q THEN
                    #testResults[13] := (#outState = 1);
                    IF #testResults[13] THEN #testPassCount := #testPassCount + 1;
                    ELSE #testFailCount := #testFailCount + 1; END_IF;
                    #testTotalSteps := #testTotalSteps + 1;
                    #tonStep(IN := FALSE, PT := T#1s);
                    #testStep := 14;
                END_IF;

            // PASO 14: Poner QT1 en LOCAL -> falla RED -> SCMTA no puede abrir QT1
            14:
                #testStatus := 'FP-14: QT1 LOCAL -> SCMTA bloqueado';
                #simDI_QT1_REMOTE_SEL := FALSE;  // LOCAL
                #simGridV_L1L2 := 200.0;
                #simGridV_L2L3 := 200.0;
                #simGridV_L3L1 := 200.0;

                #tonStep(IN := TRUE, PT := T#8s);
                IF #tonStep.Q THEN
                    // ARBITER debería bloquear el comando
                    #testResults[14] := #outBlockLocal;
                    IF #testResults[14] THEN #testPassCount := #testPassCount + 1;
                    ELSE #testFailCount := #testFailCount + 1; END_IF;
                    #testTotalSteps := #testTotalSteps + 1;
                    #tonStep(IN := FALSE, PT := T#1s);
                    #testStep := 15;
                END_IF;

            // PASO 15: Cambiar a REMOTO -> SCMTA puede continuar
            15:
                #testStatus := 'FP-15: QT1 REMOTO -> desbloquear';
                #simDI_QT1_REMOTE_SEL := TRUE;  // REMOTO

                #tonStep(IN := TRUE, PT := T#10s);
                IF #simQT1_STATE = 0 THEN
                    // QT1 se abrió (SCMTA pudo continuar)
                    #testResults[15] := TRUE;
                    #testPassCount := #testPassCount + 1;
                    #testTotalSteps := #testTotalSteps + 1;
                    #tonStep(IN := FALSE, PT := T#1s);
                    #testStep := 16;
                ELSIF #tonStep.Q THEN
                    #testResults[15] := FALSE;
                    #testFailCount := #testFailCount + 1;
                    #testTotalSteps := #testTotalSteps + 1;
                    #tonStep(IN := FALSE, PT := T#1s);
                    #testStep := 16;
                END_IF;

            // PASO 16: FAULT PATH COMPLETADO
            16:
                #testStatus := 'FP COMPLETADO - Pass:';
                #testCompleted := TRUE;
                // Reset para dejar sistema limpio
                #simGridV_L1L2 := 380.0;
                #simGridV_L2L3 := 380.0;
                #simGridV_L3L1 := 380.0;
                #simDI_QT1_REMOTE_SEL := TRUE;

        END_CASE;  // Fin FAULT PATH

    END_IF;  // Fin TEST_MODE

END_FUNCTION_BLOCK